INTERFACE I_InstanceRemovedEvent EXTENDS I_Event

PROPERTY PUBLIC Instance : I_Instance
GET
END_GET
END_PROPERTY

END_INTERFACE

(* stored: Version 1.1.0.1, ProductVersion 3.1.4024.11
   Itf I_InstanceRemovedEvent: Id {2009d3c1-018e-49dc-a886-5490f569df55}
   Property Instance: Id {4ece9284-eb60-44c9-b64d-4584b64027d3}
   Get Get: Id {42387aea-fc20-4786-bf6c-4ec9c7444e82} *)
